// ---- GlobalTextList.TcGTLO
TEXTLIST GlobalTextList
  709 = ' abort_error.error_str_1: %s'
  714 = ' abort_error.error_str_2: %s'
  705 = ' abort_error.object_name: %s'
  8 = ' CASE PACKER SHIFT REGISTERS'
  724 = ' g_application_status: %s'
  719 = ' local_ams_net_id: %s'
  1320 = ' Number Of Tasks : %i'
  1337 = ' Online Change Count : %i'
  1311 = ' Project Name : %s  '
  1328 = ' Run Time n. : %i'
  424 = '%d'
  129 = '%dxd'
  192 = '%i Insert the error to simulate'
  334 = '%i Time Exceeded'
  1303 = '%iµS [MAX]'
  1345 = '%iµS [MIN]'
  83 = '%s'
  982 = '%s Insert the error to simulate'
  247 = '1st layer robot ID'
  249 = '2nd layer robot ID'
  252 = '3rd layer robot ID'
  254 = '4th layer robot ID'
  256 = '5th layer robot ID'
  710 = '6th layer robot ID'
  677 = '< Move'
  9 = 'ACC U CHANGE'
  1429 = 'ACCU COMPLETE'
  233 = 'ACCU START POSITION REQ'
  1537 = 'ACCU START REQ'
  470 = 'Actual error: %d mm'
  694 = 'Actual error: %s mm'
  344 = 'AFL codename  %s'
  337 = 'AFL date  %s'
  339 = 'AFL version  %s'
  81 = 'aHMI present'
  78 = 'aHMI version  %s'
  663 = 'Back Stop'
  929 = 'Belts'
  317 = 'CARTESIAN MODE'
  574 = 'Carton @\nBackstop'
  181 = 'CARTON ALIGNMENT'
  415 = 'CARTON DATA MATRIX'
  921 = 'CARTON FORMING SHIFT'
  42 = 'CARTON PICKUP SHIFT'
  496 = 'Case FC Lower LS PE Covered'
  498 = 'Case FC Lower OS PE Covered'
  497 = 'Case FC Upper LS PE Covered'
  499 = 'Case FC Upper OS PE Covered'
  707 = 'Case Fed'
  1245 = 'Case Loaded'
  919 = 'Case Open Flap LS PE Covered'
  928 = 'Case Open Flap OS PE Covered'
  713 = 'Case Present'
  902 = 'Case Reject PE Status'
  675 = 'Copy >'
  77 = 'CPU Load: %i %%'
  341 = 'CPU Temp: %i °C'
  577 = 'Crosspush\nREJECT'
  575 = 'Crosspush\nRequest'
  212 = 'CUPS FEEDING SHIFT'
  572 = 'Downstream\nRedefine'
  253 = 'Downstream Backup PE Covered'
  127 = 'drum equipment'
  579 = 'dsgdd'
  581 = 'E-Stop CLOSE'
  580 = 'E-Stop OPEN'
  321 = 'Elbow: %.3f deg'
  786 = 'Emergency'
  892 = 'Emergency CLOSE'
  560 = 'Emergency CLOSED'
  342 = 'Emergency OPEN'
  495 = 'Flap Detect Photoeyes'
  466 = 'forming equipment'
  1218 = 'Glue LS Upper Flap present'
  1263 = 'Glue OS Upper Flap present'
  423 = 'has 1st layer'
  237 = 'has 2nd layer'
  239 = 'has 3rd layer'
  241 = 'has 4th layer'
  243 = 'has 5th layer'
  245 = 'has 6th layer'
  881 = 'has carton'
  809 = 'has cup'
  149 = 'has glue'
  259 = 'INCOHERENT'
  79 = 'INITIAL CONFIGURATION\n(to set before PLC Run)'
  615 = 'INNER'
  987 = 'INNER\nMISALIGNMENT'
  735 = 'Insert the error to simulate'
  6 = 'Insert the error to simulate %i'
  730 = 'Insert the error to simulate: %s mm'
  578 = 'iPhysics'
  451 = 'item rejected'
  712 = 'item to be rejected'
  513 = 'JAM'
  320 = 'JOG MINUS'
  319 = 'JOG PLUS'
  316 = 'JOINT MODE'
  469 = 'LEFT LOWER'
  343 = 'LEFT UPPER'
  508 = 'Load'
  1294 = 'load %iµS -'
  803 = 'Lower left side sensor'
  158 = 'LOWER LEFT SIDE SENSOR'
  358 = 'LOWER RIGHT SIDE SENSOR'
  1190 = 'LS Lower Flap  present'
  1227 = 'LS Open Flap  present'
  1181 = 'LS Upper Flap  present'
  829 = 'MAX'
  370 = 'MESSAGE_ aHMI_Yellow OFF'
  665 = 'MESSAGE_ aHMI_Yellow_OFF'
  845 = 'MESSAGE_aHMI_Yellow_OFF'
  384 = 'MESSAGE_aHMI_Yellow_ON'
  173 = 'MIN'
  570 = 'Move Test'
  996 = 'NOMINAL'
  936 = 'Open Flap Eyes'
  576 = 'Open Guard'
  1208 = 'OS Lower Flap  present'
  1236 = 'OS Open Flap  present'
  1199 = 'OS Upper Flap  present'
  386 = 'OUTER\nMISALIGNMENT'
  676 = 'Phase Pos: %.3f deg'
  870 = 'Phase Pos: %.3f mm'
  318 = 'PHASE REQUEST'
  992 = 'PICK CARTONS'
  822 = 'PRODUCT\nABSENCE'
  183 = 'product ID'
  251 = 'Reject Backup PE Covered'
  248 = 'Reject Present PE Covered'
  569 = 'reject reason'
  945 = 'Reject Trigger PE Covered'
  151 = 'RESET'
  652 = 'RFID'
  394 = 'RIGHT LOWER'
  3 = 'RIGHT UPPER'
  255 = 'Robot Feed'
  974 = 'Robot ID'
  80 = 'selysionare la configurazione prima di mettere RUN il PLC'
  511 = 'Shoulder: %.3f deg'
  257 = 'SHUTTLE TOGGLE'
  910 = 'Simulate Load'
  755 = 'SIMULATION EMERGENCY BUTTON'
  953 = 'SIMULATION EMERGENCY BUTTON - CASE'
  887 = 'SIMULATION EMERGENCY BUTTON - TRANSFER'
  692 = 'SIMULATION EYBOARD'
  154 = 'SIMULATION KEYBOARD'
  322 = 'Speed: %.0f deg/s'
  515 = 'Speed: %.0f mm/s'
  153 = 'START'
  169 = 'START Sim - aHMI aperto'
  674 = 'step'
  509 = 'Step 1'
  516 = 'Step 2'
  518 = 'Step 3'
  893 = 'Step 4'
  152 = 'STOP'
  700 = 'Task monitor'
  872 = 'Tilt: %.3f deg'
  1254 = 'Transfer SR1'
  61 = 'UNDER_MIN'
  464 = 'UPPER LEFT SIDE SENSOR'
  202 = 'UPPER RIGHT SIDE SENSOR'
  573 = 'Upstack\nTest\nMode'
  571 = 'Upstream\nRedefine'
  82 = 'Video presente e collegato'
  512 = 'Wrist: %.3f deg'
  514 = 'X: %.3f mm'
  871 = 'Y: %.3f mm'
  88 = 'Yellow Message OFF'
  771 = 'Yellow Message ON'
  729 = '[1] highest %iµS - '
  734 = '[2] norm %iµS - '
  1277 = '[3] low %iµS - '
  1286 = '[4] lowest %iµS - '
END_TEXTLIST

// ---- Visualization/AFL/VISU_MAIN.TcVIS
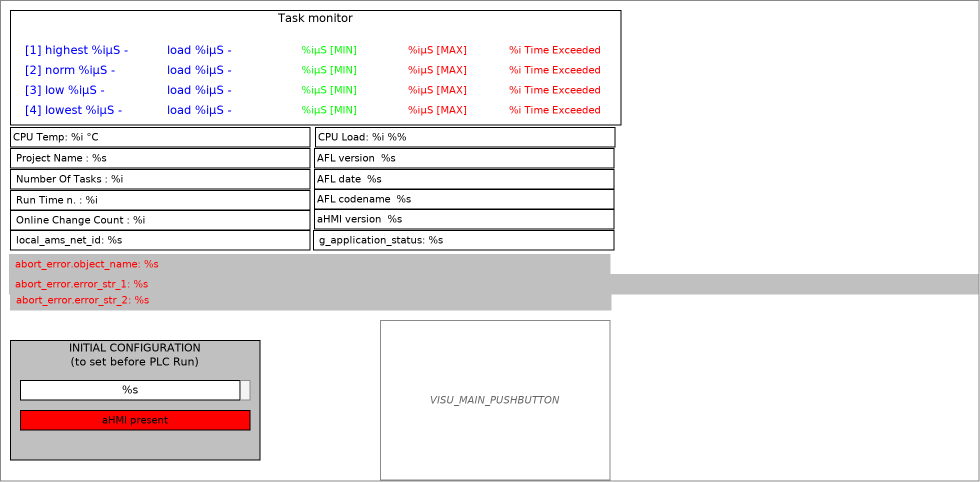
VISUALIZATION VISU_MAIN  // 980x482
    Rectangle (10,10 611x115), "Task monitor"
    Rectangle (9,254 601x20), "abort_error.object_name: %s", text variable: abort_error.object_name
    Rectangle (9,274 969x20), "abort_error.error_str_1: %s", text variable: abort_error.error_str_1
    Rectangle (10,290 601x20), "abort_error.error_str_2: %s", text variable: abort_error.error_str_2
    Rectangle (10,230 300x20), "local_ams_net_id: %s", text variable: local_ams_net_id
    Rectangle (313,230 301x20), "g_application_status: %s", text variable: Application_Common.g_application_status
    Rectangle (22,40 130x20), "[1] highest %iµS -", text variable: afl_tasks[1].cycle_us
    Rectangle (22,60 130x20), "[2] norm %iµS -", text variable: afl_tasks[2].cycle_us
    Rectangle (22,80 130x20), "[3] low %iµS -", text variable: afl_tasks[3].cycle_us
    Rectangle (22,100 130x20), "[4] lowest %iµS -", text variable: afl_tasks[4].cycle_us
    Rectangle (164,100 100x20), "load %iµS -", text variable: afl_tasks[4].task_profiler_data.AverageExecTime
    Rectangle (164,80 100x20), "load %iµS -", text variable: afl_tasks[3].task_profiler_data.AverageExecTime
    Rectangle (164,60 100x20), "load %iµS -", text variable: afl_tasks[2].task_profiler_data.AverageExecTime
    Rectangle (164,40 100x20), "load %iµS -", text variable: afl_tasks[1].task_profiler_data.AverageExecTime
    Rectangle (380,40 90x20), "%iµS [MAX]", text variable: afl_tasks[1].task_profiler_data.MaxExecTime
    Rectangle (380,60 90x20), "%iµS [MAX]", text variable: afl_tasks[2].task_profiler_data.MaxExecTime
    Rectangle (380,80 90x20), "%iµS [MAX]", text variable: afl_tasks[2].task_profiler_data.MaxExecTime
    Rectangle (380,100 90x20), "%iµS [MAX]", text variable: afl_tasks[4].task_profiler_data.MaxExecTime
    Rectangle (10,148 300x20), "Project Name : %s", text variable: SystemInfo.projectName
    Rectangle (10,169 300x20), "Number Of Tasks : %i", text variable: SystemInfo.numberOfTasks
    Rectangle (10,190 300x20), "Run Time n. : %i", text variable: SystemInfo.runTimeNo
    Rectangle (10,210 300x20), "Online Change Count : %i", text variable: SystemInfo.onlineChangeCount
    Rectangle (250,100 110x20), "%iµS [MIN]", text variable: afl_tasks[4].task_profiler_data.MinExecTime
    Rectangle (250,80 110x20), "%iµS [MIN]", text variable: afl_tasks[3].task_profiler_data.MinExecTime
    Rectangle (250,60 110x20), "%iµS [MIN]", text variable: afl_tasks[2].task_profiler_data.MinExecTime
    Rectangle (250,40 110x20), "%iµS [MIN]", text variable: afl_tasks[1].task_profiler_data.MinExecTime
    Rectangle (506,40 110x20), "%i Time Exceeded", text variable: SystemTaskInfoArr[1].cycleTimeExceeded
    Rectangle (506,60 110x20), "%i Time Exceeded", text variable: SystemTaskInfoArr[2].cycleTimeExceeded
    Rectangle (506,80 110x20), "%i Time Exceeded", text variable: SystemTaskInfoArr[3].cycleTimeExceeded
    Rectangle (506,100 110x20), "%i Time Exceeded", text variable: SystemTaskInfoArr[4].cycleTimeExceeded
    Rectangle (314,169 300x20), "AFL date %s", text variable: AFL_VERSION.v_date
    Rectangle (314,148 300x20), "AFL version %s", text variable: AFL_VERSION.s_value
    Rectangle (10,127 300x20), "CPU Temp: %i °C", text variable: .system_diagnosis.cpu_temperature_actual_value
    Rectangle (314,189 300x20), "AFL codename %s", text variable: AFL_VERSION.development_stage
    Rectangle (315,127 300x20), "CPU Load: %i %%", text variable: system_diagnosis.cpu_usage_actual_value
    Rectangle (314,209 300x20), "aHMI version %s", text variable: hmi.private.major_version
    Frame (380,320 230x160)
        shows VISU_MAIN_PUSHBUTTON(m_Input_mch := EZ.mch, m_Input_stop := ez_mch_services_pushbuttons_main.stop_button_di, m_Input_reset := ez_mch_services_pushbuttons_main.reset_button_di, m_Input_start := ez_mch_services_pushbuttons_main.start_button_pressed_di)
    Rectangle (10,340 250x120), "INITIAL CONFIGURATION (to set before PLC Run)", tooltip "selysionare la configurazione prima di mettere RUN il PLC"
    RoundedRectangle (20,410 230x20), "aHMI present", tooltip "Video presente e collegato", colour toggle: Application_Common.HMI_IS_REQUIRED_DVR
        toggle Application_Common.HMI_IS_REQUIRED_DVR
    RoundedRectangle (20,380 220x20), "%s", text variable: .test_target_device
    Scrollbar (240,380 10x20)
        p1057716461: .test_target_device
END_VISUALIZATION

// ---- Visualization/Carton feeding/CARTON_FEEDING_TOOTH_DISTANCE.TcVIS
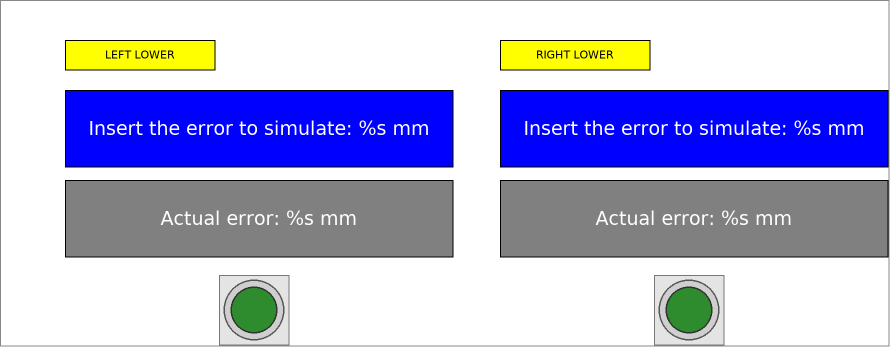
VISUALIZATION CARTON_FEEDING_TOOTH_DISTANCE  // 890x347
    Rectangle (65,40 150x30), "LEFT LOWER"
    Rectangle (500,40 150x30), "RIGHT LOWER"
    RoundedRectangle (65,90 388x77), "Insert the error to simulate: %s mm", text variable: wu_cartonFeeding_leftSide_toothDistance.simulation_error
        OnMouseUp: write the text variable via VisuDialogs.Numpad
    RoundedRectangle (500,90 388x77), "Insert the error to simulate: %s mm", text variable: wu_cartonFeeding_rightSide_toothDistance.simulation_error
        OnMouseUp: write the text variable via VisuDialogs.Numpad
    RoundedRectangle (65,180 388x77), "Actual error: %s mm", text variable: wu_cartonFeeding_leftSide_toothDistance.simulation_error_current_value_visu
        OnMouseUp: write the text variable via VisuDialogs.Numpad
    RoundedRectangle (500,180 388x77), "Actual error: %s mm", text variable: wu_cartonFeeding_rightSide_toothDistance.simulation_error_current_value_visu
        OnMouseUp: write the text variable via VisuDialogs.Numpad
    PushSwitch (219,275 70x70), variable: wu_cartonFeeding_leftSide_toothDistance.simulation_error_download, behaviour: TAP, style: Switch-PushSwitch-Green
    PushSwitch (654,275 70x70), variable: wu_cartonFeeding_rightSide_toothDistance.simulation_error_download, behaviour: TAP, style: Switch-PushSwitch-Green
END_VISUALIZATION

// ---- Visualization/Carton forming/CARTON_FORMING_CHECKS.TcVIS
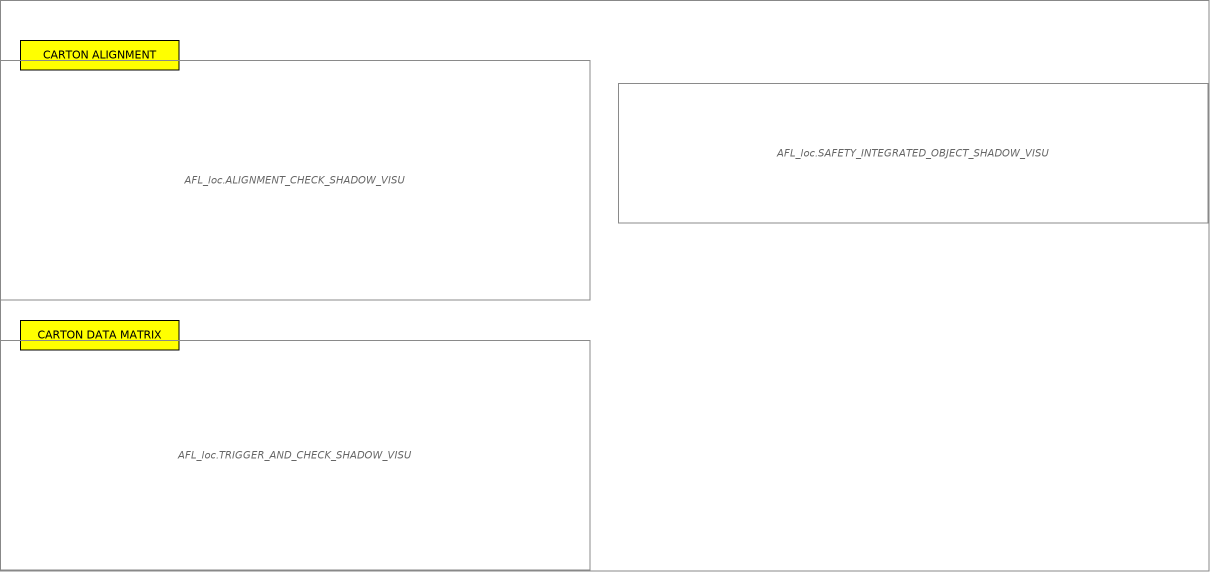
VISUALIZATION CARTON_FORMING_CHECKS  // 1210x572
    Rectangle (20,40 159x30), "CARTON ALIGNMENT"
    Frame (0,60 590x240)
        shows AFL_loc.ALIGNMENT_CHECK_SHADOW_VISU(m_Input_alignment_check_shadow := dbg_wu_cartonforming_belt_checks.algnchk_shd)
    Rectangle (20,320 159x30), "CARTON DATA MATRIX"
    Frame (0,340 590x230)
        shows AFL_loc.TRIGGER_AND_CHECK_SHADOW_VISU(m_Input_trigger_and_check_shadow := dbg_wu_cartonforming_belt_checks.data_matrix_tchk_shd)
    Frame (618,83 590x140)
        shows AFL_loc.SAFETY_INTEGRATED_OBJECT_SHADOW_VISU(m_Input_safety_integrated_object_shadow := dbg_wu_main_safety_guards.sio_shd)
END_VISUALIZATION

// ---- Visualization/Casepacker_Keyboard.TcVIS
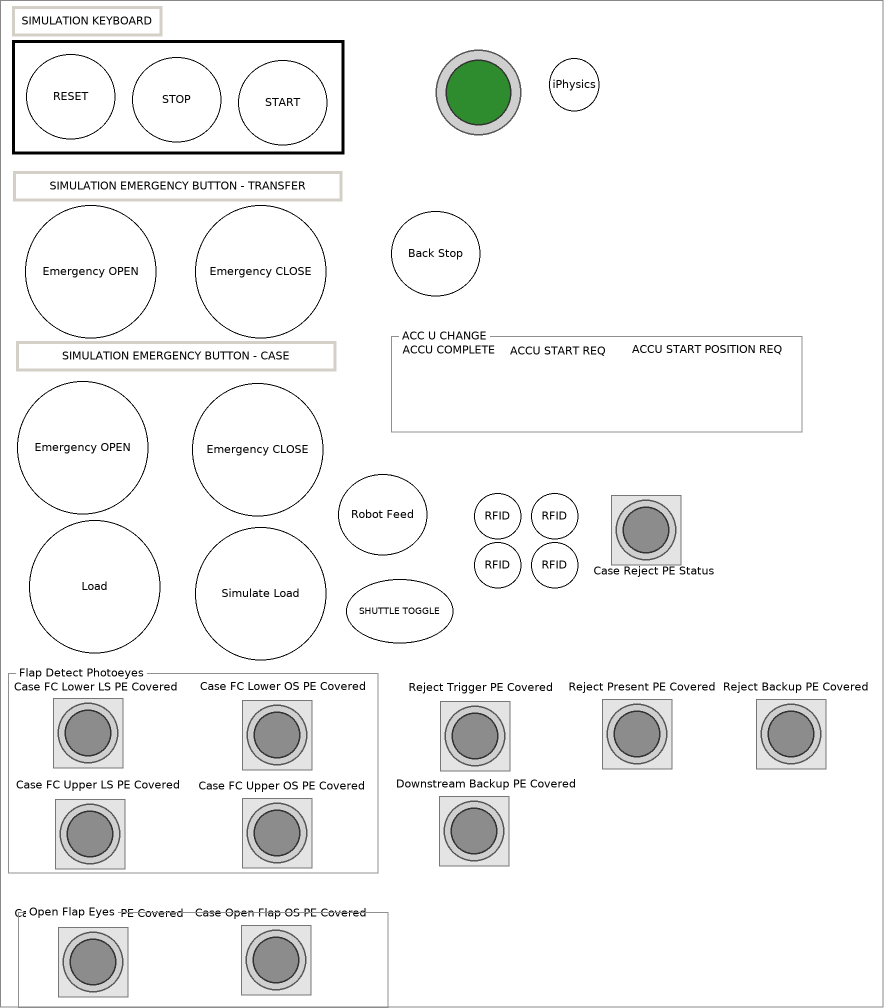
VISUALIZATION Casepacker_Keyboard  // 884x1008
    Rectangle (12,40 332x114)
    Ellipse (26,54 89x85), "RESET"
        tap csp_transfer_main_services_pushbuttons.visu_reset
    Ellipse (132,57 89x85), "STOP"
        tap csp_transfer_main_services_pushbuttons.visu_stop
    Ellipse (238,60 89x85), "START"
        tap csp_transfer_main_services_pushbuttons.visu_start
    Textfield (12,6 150x30), "SIMULATION KEYBOARD"
    Ellipse (25,205 131x133), "Emergency OPEN"
        tap csp_transfer_main_services_pushbuttons.visu_emergency_open
    Ellipse (195,205 131x133), "Emergency CLOSE"
        tap csp_transfer_main_services_pushbuttons.visu_emergency_close
    Textfield (13,171 329x30), "SIMULATION EMERGENCY BUTTON - TRANSFER"
    Lamp1 (426,43 105x99), variable: csp_transfer_main_safety_emergency.HMI_button_lamp_do.field.status, style: Lamp-Lamp1-Green
    Ellipse (391,211 89x85), "Back Stop", colour toggle: csp_transfer_upstacker_sensors.debug_carton_backstop
        toggle csp_transfer_upstacker_sensors.debug_carton_backstop
    Ellipse (192,383 131x133), "Emergency CLOSE"
        tap csp_case_main_services_pushbuttons.visu_emergency_close
    Textfield (16,341 320x30), "SIMULATION EMERGENCY BUTTON - CASE"
    Ellipse (17,381 131x133), "Emergency OPEN"
        tap csp_case_main_services_pushbuttons.visu_emergency_open
    Ellipse (549,58 50x53), "iPhysics"
        toggle MAIN.IP_enable
    GroupBox (8,665 370x208), "Flap Detect Photoeyes"
        PushSwitchLed (45,33 70x70), variable: dbg_csp_case_fc_ls_lower_sensors.flap_chksect_shd.force_input_status, behaviour: TOGGLE, style: Switch-PushSwitchLed-Gray
    Ellipse (29,520 131x133), "Load"
        tap csp_case_loader.load_request
    Ellipse (531,493 47x46), "RFID"
        toggle csp_case_closing_ls_upper.rfid_fake
    Ellipse (531,542 47x46), "RFID"
        toggle csp_case_closing_ls_lower.rfid_fake
    Ellipse (474,493 47x46), "RFID"
        toggle csp_case_closing_os_upper.rfid_fake
    Ellipse (474,542 47x46), "RFID"
        toggle csp_case_closing_os_lower.rfid_fake
    PushSwitchLed (611,495 70x70), behaviour: TOGGLE, style: Switch-PushSwitchLed-Gray
    Label (579,556 150x30), "Case Reject PE Status"
    Ellipse (195,527 131x133), "Simulate Load"
        tap csp_case_transport.product_loaded
    Label (8,673 176x28), "Case FC Lower LS PE Covered"
    PushSwitchLed (55,799 70x70), variable: dbg_csp_case_fc_ls_upper_sensors.flap_chksect_shd.force_input_status, behaviour: TOGGLE, style: Switch-PushSwitchLed-Gray
    Label (10,775 176x20), "Case FC Upper LS PE Covered"
    PushSwitchLed (242,700 70x70), variable: dbg_csp_case_fc_os_lower_sensors.flap_chksect_shd.force_input_status, behaviour: TOGGLE, style: Switch-PushSwitchLed-Gray
    Label (195,678 176x17), "Case FC Lower OS PE Covered"
    PushSwitchLed (242,798 70x70), variable: dbg_csp_case_fc_os_upper_sensors.flap_chksect_shd.force_input_status, behaviour: TOGGLE, style: Switch-PushSwitchLed-Gray
    Label (194,777 176x18), "Case FC Upper OS PE Covered"
    Label (8,888 176x28)
    PushSwitchLed (58,927 70x70), variable: dbg_csp_case_openflap_sensors.open_flap_ls_di_dchk_shd.force_input_status, behaviour: TOGGLE, style: Switch-PushSwitchLed-Gray
    Label (11,905 176x17), "Case Open Flap LS PE Covered"
    PushSwitchLed (241,925 70x70), variable: dbg_csp_case_openflap_sensors.open_flap_os_di_dchk_shd.force_input_status, behaviour: TOGGLE, style: Switch-PushSwitchLed-Gray
    Label (193,904 176x18), "Case Open Flap OS PE Covered"
    GroupBox (391,328 411x104), "ACC U CHANGE"
        Label (381,-232 176x28)
        Label (79,9 176x28), "ACCU START REQ"
    PushSwitchLed (440,701 70x70), variable: dbg_csp_case_discharge_reject_sensors.reject_trigger_inchoerence_chksect_shd.force_input_status, behaviour: TOGGLE, style: Switch-PushSwitchLed-Gray
    Label (393,679 176x17), "Reject Trigger PE Covered"
    PushSwitchLed (602,699 70x70), variable: dbg_csp_case_discharge_reject_sensors.reject_present_di_shd.is_covered, behaviour: TOGGLE, style: Switch-PushSwitchLed-Gray
    Label (554,678 176x18), "Reject Present PE Covered"
    PushSwitchLed (756,699 70x70), variable: dbg_csp_case_discharge_reject_sensors.reject_backup_di_shd.is_covered, behaviour: TOGGLE, style: Switch-PushSwitchLed-Gray
    Label (708,678 176x18), "Reject Backup PE Covered"
    PushSwitchLed (439,796 70x70), variable: dbg_csp_case_discharge_reject_sensors.downstream_backup_di_shd.is_covered, behaviour: TOGGLE, style: Switch-PushSwitchLed-Gray
    Label (391,775 190x18), "Downstream Backup PE Covered"
    Ellipse (338,474 89x81), "Robot Feed"
        toggle csp_case_feed.Feed_request
    Ellipse (346,579 107x64), "SHUTTLE TOGGLE"
        toggle csp_case_transport.product_loaded
    GroupBox (18,904 370x104), "Open Flap Eyes"
        Label (381,-232 176x28)
    Label (361,336 176x28), "ACCU COMPLETE"
    Label (619,327 176x45), "ACCU START POSITION REQ"
END_VISUALIZATION

// ---- Visualization/cp_visu/Visualization_1.TcVIS
VISUALIZATION Visualization_1  // 2x2
END_VISUALIZATION

// ---- Visualization/CSP_Case_Feed_Kinematic.TcVIS
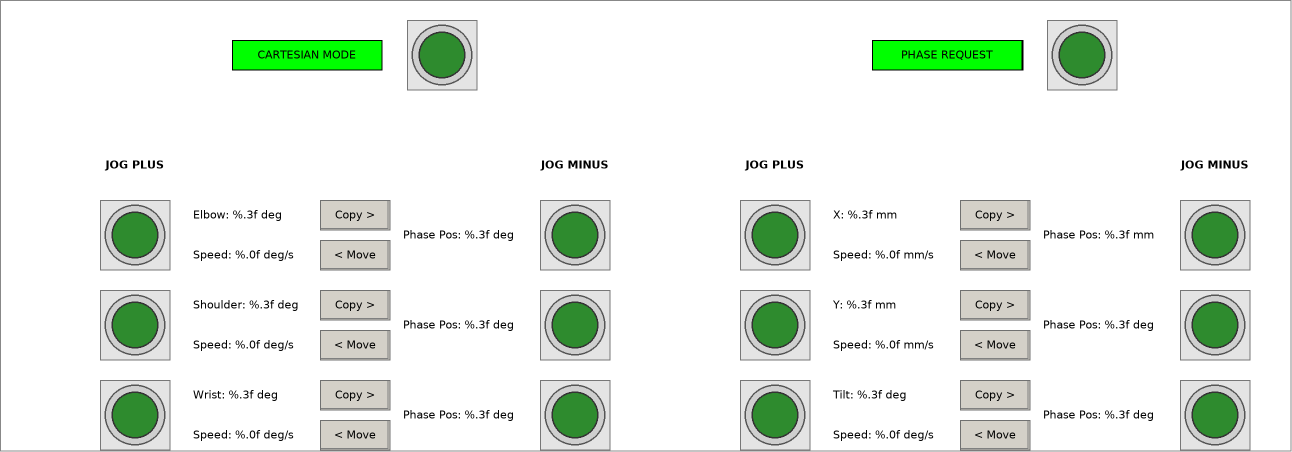
VISUALIZATION CSP_Case_Feed_Kinematic  // 1292x452
    Group (232,20 245x70)
        Rectangle (0,20 150x30), "JOINT MODE", invisible if: csp_case_feed_kinematic.kin_config_cartesian_mode
        PushSwitch (175,0 70x70), variable: csp_case_feed_kinematic.joint_cartesian_mode, input disabled if: csp_case_feed_kinematic.visu_disable_general_command, behaviour: TAP, style: Switch-PushSwitch-Green
        Rectangle (0,20 150x30), "CARTESIAN MODE", invisible if: not csp_case_feed_kinematic.kin_config_cartesian_mode
    Group (872,20 245x70)
        Rectangle (1,20 150x30), "PHASE REQUEST", invisible if: csp_case_feed_kinematic.phase_request
        PushSwitch (175,0 70x70), variable: csp_case_feed_kinematic.phase_request, input disabled if: csp_case_feed_kinematic.visu_disable_phase_request, behaviour: TOGGLE, style: Switch-PushSwitch-Green
        Rectangle (0,20 150x30), "PHASE REQUEST", invisible if: not csp_case_feed_kinematic.phase_request
    Rectangle (60,150 150x30), "JOG PLUS"
    Rectangle (500,150 150x30), "JOG MINUS"
    Group (100,200 510x70)
        Rectangle (90,0 140x30), "Elbow: %.3f deg", text variable: csp_case_feed_kinematic.elbow_actual_position
        PushSwitch (0,0 70x70), variable: csp_case_feed_kinematic.elbow_jog_plus, input disabled if: csp_case_feed_kinematic.visu_disable_ACS_jog_mode, behaviour: TAP, style: Switch-PushSwitch-Green
        PushSwitch (440,0 70x70), variable: csp_case_feed_kinematic.elbow_jog_minus, input disabled if: csp_case_feed_kinematic.visu_disable_ACS_jog_mode, behaviour: TAP, style: Switch-PushSwitch-Green
        Rectangle (90,40 140x30), "Speed: %.0f deg/s", text variable: csp_case_feed_kinematic.elbow_move_speed
            OnMouseDown: write csp_case_feed_kinematic.elbow_move_speed via VisuDialogs.Numpad, min 0, max 100, format %.0f
        Button (220,0 70x30), "Copy >", input disabled if: csp_case_feed_kinematic.visu_disable_ACS_command
            tap csp_case_feed_kinematic.elbow_copy_phase
        Rectangle (300,20 140x30), "Phase Pos: %.3f deg", text variable: csp_case_feed_kinematic.elbow_phase_position
            OnMouseDown: write csp_case_feed_kinematic.elbow_phase_position via VisuDialogs.Numpad, min -200, max 200, format %.3f
        Button (220,40 70x30), "< Move", input disabled if: csp_case_feed_kinematic.visu_disable_ACS_command
            tap csp_case_feed_kinematic.elbow_phase_move
    Group (100,290 510x70)
        Rectangle (90,0 140x30), "Shoulder: %.3f deg", text variable: csp_case_feed_kinematic.shoulder_actual_position
        PushSwitch (0,0 70x70), variable: csp_case_feed_kinematic.shoulder_jog_plus, input disabled if: csp_case_feed_kinematic.visu_disable_ACS_jog_mode, behaviour: TAP, style: Switch-PushSwitch-Green
        PushSwitch (440,0 70x70), variable: csp_case_feed_kinematic.shoulder_jog_minus, input disabled if: csp_case_feed_kinematic.visu_disable_ACS_jog_mode, behaviour: TAP, style: Switch-PushSwitch-Green
        Rectangle (90,40 140x30), "Speed: %.0f deg/s", text variable: csp_case_feed_kinematic.shoulder_move_speed
            OnMouseDown: write csp_case_feed_kinematic.shoulder_move_speed via VisuDialogs.Numpad, min 0, max 100, format %.0f
        Button (220,0 70x30), "Copy >", input disabled if: csp_case_feed_kinematic.visu_disable_ACS_command
            tap csp_case_feed_kinematic.shoulder_copy_phase
        Rectangle (300,20 140x30), "Phase Pos: %.3f deg", text variable: csp_case_feed_kinematic.shoulder_phase_position
            OnMouseDown: write csp_case_feed_kinematic.shoulder_phase_position via VisuDialogs.Numpad, min -200, max 200, format %.3f
        Button (220,40 70x30), "< Move", input disabled if: csp_case_feed_kinematic.visu_disable_ACS_command
            tap csp_case_feed_kinematic.shoulder_phase_move
    Group (100,380 510x70)
        Rectangle (90,0 140x30), "Wrist: %.3f deg", text variable: csp_case_feed_kinematic.wrist_actual_position
        PushSwitch (0,0 70x70), variable: csp_case_feed_kinematic.wrist_jog_plus, input disabled if: csp_case_feed_kinematic.visu_disable_ACS_jog_mode, behaviour: TAP, style: Switch-PushSwitch-Green
        PushSwitch (440,0 70x70), variable: csp_case_feed_kinematic.wrist_jog_minus, input disabled if: csp_case_feed_kinematic.visu_disable_ACS_jog_mode, behaviour: TAP, style: Switch-PushSwitch-Green
        Rectangle (90,40 140x30), "Speed: %.0f deg/s", text variable: csp_case_feed_kinematic.wrist_move_speed
            OnMouseDown: write csp_case_feed_kinematic.wrist_move_speed via VisuDialogs.Numpad, min 0, max 100, format %.0f
        Button (220,0 70x30), "Copy >", input disabled if: csp_case_feed_kinematic.visu_disable_ACS_command
            tap csp_case_feed_kinematic.wrist_copy_phase
        Rectangle (300,20 140x30), "Phase Pos: %.3f deg", text variable: csp_case_feed_kinematic.wrist_phase_position
            OnMouseDown: write csp_case_feed_kinematic.wrist_phase_position via VisuDialogs.Numpad, min -200, max 200, format %.3f
        Button (220,40 70x30), "< Move", input disabled if: csp_case_feed_kinematic.visu_disable_ACS_command
            tap csp_case_feed_kinematic.wrist_phase_move
    Group (740,200 510x70)
        Rectangle (90,0 140x30), "X: %.3f mm", text variable: csp_case_feed_kinematic.x_actual_position
        PushSwitch (0,0 70x70), variable: csp_case_feed_kinematic.x_jog_plus, input disabled if: csp_case_feed_kinematic.visu_disable_MCS_jog_mode, behaviour: TAP, style: Switch-PushSwitch-Green
        PushSwitch (440,0 70x70), variable: csp_case_feed_kinematic.x_jog_minus, input disabled if: csp_case_feed_kinematic.visu_disable_MCS_jog_mode, behaviour: TAP, style: Switch-PushSwitch-Green
        Rectangle (90,40 140x30), "Speed: %.0f mm/s", text variable: csp_case_feed_kinematic.x_move_speed
            OnMouseDown: write csp_case_feed_kinematic.x_move_speed via VisuDialogs.Numpad, min 0, max 100, format %.0f
        Button (220,0 70x30), "Copy >", input disabled if: csp_case_feed_kinematic.visu_disable_MCS_command
            tap csp_case_feed_kinematic.x_copy_phase
        Rectangle (300,20 140x30), "Phase Pos: %.3f mm", text variable: csp_case_feed_kinematic.x_phase_position
            OnMouseDown: write csp_case_feed_kinematic.x_phase_position via VisuDialogs.Numpad, min -2000, max 2000, format %.3f
        Button (220,40 70x30), "< Move", input disabled if: csp_case_feed_kinematic.visu_disable_MCS_command
            tap csp_case_feed_kinematic.x_phase_move
    Rectangle (1140,150 150x30), "JOG MINUS"
    Rectangle (700,150 150x30), "JOG PLUS"
    Group (740,290 510x70)
        Rectangle (90,0 140x30), "Y: %.3f mm", text variable: csp_case_feed_kinematic.y_actual_position
        PushSwitch (0,0 70x70), variable: csp_case_feed_kinematic.y_jog_plus, input disabled if: csp_case_feed_kinematic.visu_disable_MCS_jog_mode, behaviour: TAP, style: Switch-PushSwitch-Green
        PushSwitch (440,0 70x70), variable: csp_case_feed_kinematic.y_jog_minus, input disabled if: csp_case_feed_kinematic.visu_disable_MCS_jog_mode, behaviour: TAP, style: Switch-PushSwitch-Green
        Rectangle (90,40 140x30), "Speed: %.0f mm/s", text variable: csp_case_feed_kinematic.y_move_speed
            OnMouseDown: write csp_case_feed_kinematic.y_move_speed via VisuDialogs.Numpad, min 0, max 100, format %.0f
        Button (220,0 70x30), "Copy >", input disabled if: csp_case_feed_kinematic.visu_disable_MCS_command
            tap csp_case_feed_kinematic.y_copy_phase
        Rectangle (300,20 140x30), "Phase Pos: %.3f deg", text variable: csp_case_feed_kinematic.y_phase_position
            OnMouseDown: write csp_case_feed_kinematic.y_phase_position via VisuDialogs.Numpad, min -100, max 1000, format %.3f
        Button (220,40 70x30), "< Move", input disabled if: csp_case_feed_kinematic.visu_disable_MCS_command
            tap csp_case_feed_kinematic.y_phase_move
    Group (740,380 510x70)
        Rectangle (90,0 140x30), "Tilt: %.3f deg", text variable: csp_case_feed_kinematic.tilt_actual_position
        PushSwitch (0,0 70x70), variable: csp_case_feed_kinematic.tilt_jog_plus, input disabled if: csp_case_feed_kinematic.visu_disable_MCS_jog_mode, behaviour: TAP, style: Switch-PushSwitch-Green
        PushSwitch (440,0 70x70), variable: csp_case_feed_kinematic.tilt_jog_minus, input disabled if: csp_case_feed_kinematic.visu_disable_MCS_jog_mode, behaviour: TAP, style: Switch-PushSwitch-Green
        Rectangle (90,40 140x30), "Speed: %.0f deg/s", text variable: csp_case_feed_kinematic.tilt_move_speed
            OnMouseDown: write csp_case_feed_kinematic.tilt_move_speed via VisuDialogs.Numpad, min 0, max 100, format %.0f
        Button (220,0 70x30), "Copy >", input disabled if: csp_case_feed_kinematic.visu_disable_MCS_command
            tap csp_case_feed_kinematic.tilt_copy_phase
        Rectangle (300,20 140x30), "Phase Pos: %.3f deg", text variable: csp_case_feed_kinematic.tilt_phase_position
            OnMouseDown: write csp_case_feed_kinematic.tilt_phase_position via VisuDialogs.Numpad, min 0, max 150, format %.3f
        Button (220,40 70x30), "< Move", input disabled if: csp_case_feed_kinematic.visu_disable_MCS_command
            tap csp_case_feed_kinematic.tilt_phase_move
END_VISUALIZATION

// ---- Visualization/Transfer_Keyboard.TcVIS
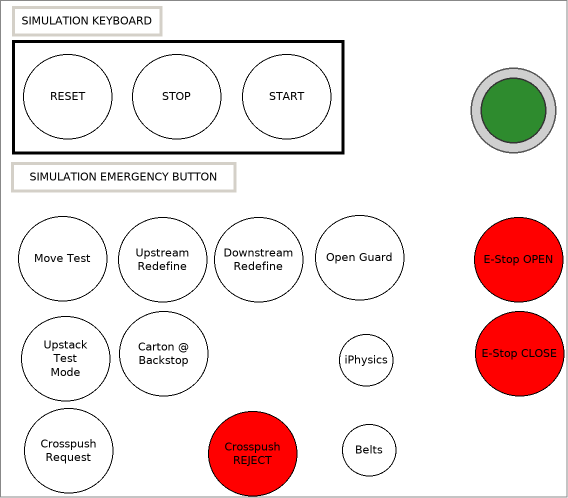
VISUALIZATION Transfer_Keyboard  // 568x498
    Rectangle (12,40 332x114)
    Ellipse (23,54 89x85), "RESET"
        tap csp_transfer_main_services_pushbuttons.visu_reset
    Ellipse (132,54 89x85), "STOP"
        tap csp_transfer_main_services_pushbuttons.visu_stop
    Ellipse (242,54 89x85), "START"
        tap csp_transfer_main_services_pushbuttons.visu_start
    Textfield (12,6 150x30), "SIMULATION KEYBOARD"
    Textfield (11,162 225x30), "SIMULATION EMERGENCY BUTTON"
    Lamp1 (461,61 105x99), variable: csp_transfer_main_safety_emergency.HMI_button_lamp_do.field.status, style: Lamp-Lamp1-Green
    Ellipse (18,216 89x85), "Move Test"
        toggle csp_transfer_upstacker_virtualMaster.move_test_enable
    Ellipse (118,217 89x85), "Upstream Redefine"
        tap csp_transfer_upstacker_virtualMaster.move_test_redefine_upstream
    Ellipse (214,217 89x85), "Downstream Redefine"
        tap csp_transfer_upstacker_virtualMaster.move_test_redefine_downstream
    Ellipse (21,316 89x85), "Upstack Test Mode"
        toggle csp_transfer_upstacker_sensors.debug_active
    Ellipse (119,311 89x85), "Carton @ Backstop"
        toggle csp_transfer_upstacker_sensors.debug_carton_backstop
    Ellipse (24,408 89x85), "Crosspush Request"
        toggle csp_transfer_crosspusher.move_request
    Ellipse (315,215 89x85), "Open Guard"
        toggle csp_transfer_upstacker_virtualMaster.guard_open
    Ellipse (208,411 89x85), "Crosspush REJECT"
        tap csp_transfer_crosspusher_sensors.reject_stack
    Ellipse (339,334 54x52), "iPhysics"
        toggle IP_Main.IP_enable
    Ellipse (474,217 89x85), "E-Stop OPEN"
        tap csp_case_main_services_pushbuttons.visu_emergency_open
    Ellipse (475,311 89x85), "E-Stop CLOSE"
        tap csp_case_main_services_pushbuttons.visu_emergency_close
    Ellipse (342,424 54x52), "Belts"
        toggle csp_transfer_infeed_clamp.start_infeed_belts
END_VISUALIZATION

// ---- Visualization/Shift register/Carton filling/CARTON_FILLING_SHIFT_ELEMENT.TcVIS
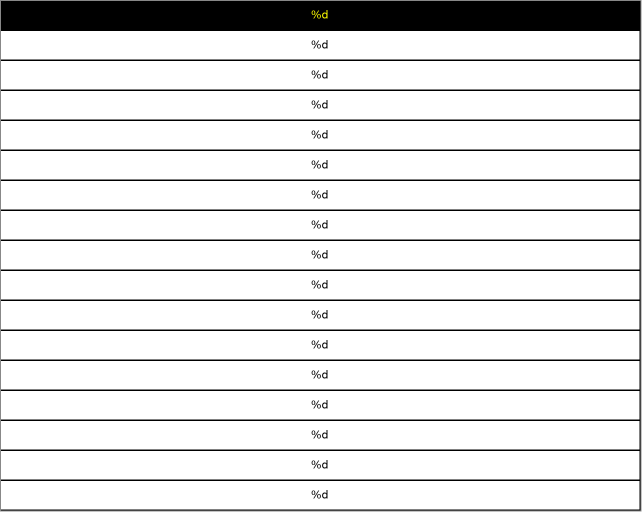
VISUALIZATION CARTON_FILLING_SHIFT_ELEMENT  // 642x512
VAR_INPUT
	index:		UDINT;
END_VAR
    Rectangle (0,0 640x30), "%d", text variable: wu_cartonForming_shiftRegister_debug.shift_debug[index].step_id
    Rectangle (0,30 640x30), "%d", text variable: wu_cartonFilling_shiftRegister_debug.shift_debug[index].status.0, colour toggle: wu_cartonFilling_shiftRegister_debug.shift_debug[index].status.0
    Rectangle (0,90 640x30), "%d", text variable: wu_cartonFilling_shiftRegister_debug.shift_debug[index].reject_reason
    Rectangle (0,120 640x30), "%d", text variable: wu_cartonFilling_shiftRegister_debug.shift_debug[index].status.4, colour toggle: wu_cartonFilling_shiftRegister_debug.shift_debug[index].status.4
    Rectangle (0,180 640x30), "%d", text variable: wu_cartonFilling_shiftRegister_debug.shift_debug[index].status.11, colour toggle: wu_cartonFilling_shiftRegister_debug.shift_debug[index].status.11
    Rectangle (0,150 640x30), "%d", text variable: wu_cartonFilling_shiftRegister_debug.shift_debug[index].status.10, colour toggle: wu_cartonFilling_shiftRegister_debug.shift_debug[index].status.10
    Rectangle (0,60 640x30), "%d", text variable: wu_cartonFilling_shiftRegister_debug.shift_debug[index].status.1, colour toggle: wu_cartonFilling_shiftRegister_debug.shift_debug[index].status.1
    Rectangle (0,210 640x30), "%d", text variable: wu_cartonFilling_shiftRegister_debug.shift_debug[index].status.12, colour toggle: wu_cartonFilling_shiftRegister_debug.shift_debug[index].status.12
    Rectangle (0,240 640x30), "%d", text variable: wu_cartonFilling_shiftRegister_debug.shift_debug[index].status.13, colour toggle: wu_cartonFilling_shiftRegister_debug.shift_debug[index].status.13
    Rectangle (0,270 640x30), "%d", text variable: wu_cartonFilling_shiftRegister_debug.shift_debug[index].status.14, colour toggle: wu_cartonFilling_shiftRegister_debug.shift_debug[index].status.14
    Rectangle (0,300 640x30), "%d", text variable: wu_cartonFilling_shiftRegister_debug.shift_debug[index].status.15, colour toggle: wu_cartonFilling_shiftRegister_debug.shift_debug[index].status.15
    Rectangle (0,330 640x30), "%d", text variable: wu_cartonFilling_shiftRegister_debug.shift_debug[index]._1st_layer_robot_id
    Rectangle (0,360 640x30), "%d", text variable: wu_cartonFilling_shiftRegister_debug.shift_debug[index]._2nd_layer_robot_id
    Rectangle (0,390 640x30), "%d", text variable: wu_cartonFilling_shiftRegister_debug.shift_debug[index]._3rd_layer_robot_id
    Rectangle (0,420 640x30), "%d", text variable: wu_cartonFilling_shiftRegister_debug.shift_debug[index]._4th_layer_robot_id
    Rectangle (0,450 640x30), "%d", text variable: wu_cartonFilling_shiftRegister_debug.shift_debug[index]._5th_layer_robot_id
    Rectangle (0,480 640x30), "%d", text variable: wu_cartonFilling_shiftRegister_debug.shift_debug[index]._6th_layer_robot_id
END_VISUALIZATION

// ---- Visualization/Shift register/Carton filling/CARTON_FILLING_SHIFT_ELEMENT_DESCRIPTION.TcVIS
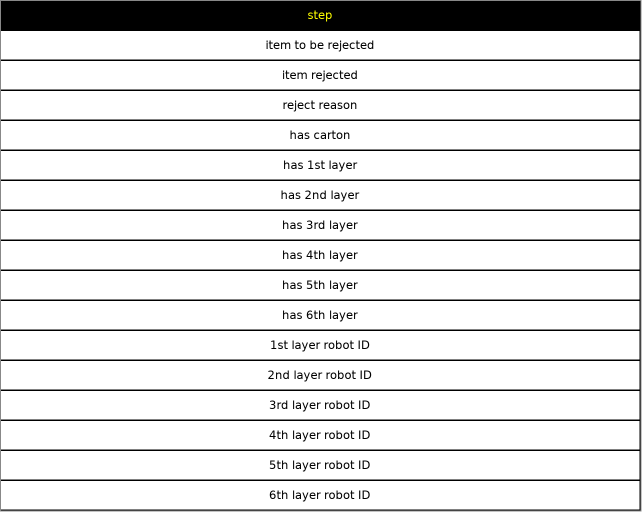
VISUALIZATION CARTON_FILLING_SHIFT_ELEMENT_DESCRIPTION  // 642x512
    Rectangle (0,0 640x30), "step"
    Rectangle (0,30 640x30), "item to be rejected"
    Rectangle (0,90 640x30), "reject reason"
    Rectangle (0,120 640x30), "has carton"
    Rectangle (0,150 640x30), "has 1st layer"
    Rectangle (0,60 640x30), "item rejected"
    Rectangle (0,180 640x30), "has 2nd layer"
    Rectangle (0,210 640x30), "has 3rd layer"
    Rectangle (0,240 640x30), "has 4th layer"
    Rectangle (0,270 640x30), "has 5th layer"
    Rectangle (0,300 640x30), "has 6th layer"
    Rectangle (0,330 640x30), "1st layer robot ID"
    Rectangle (0,360 640x30), "2nd layer robot ID"
    Rectangle (0,390 640x30), "3rd layer robot ID"
    Rectangle (0,420 640x30), "4th layer robot ID"
    Rectangle (0,450 640x30), "5th layer robot ID"
    Rectangle (0,480 640x30), "6th layer robot ID"
END_VISUALIZATION

// ---- Visualization/Shift register/Carton forming/CARTON_FORMING_SHIFT_ELEMENT.TcVIS
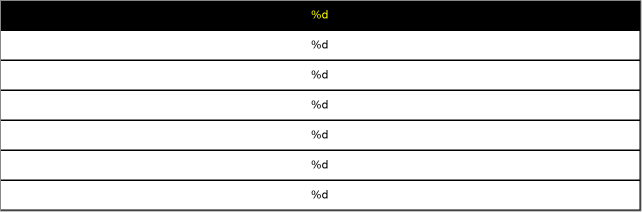
VISUALIZATION CARTON_FORMING_SHIFT_ELEMENT  // 642x212
VAR_INPUT
	index:		UDINT;
END_VAR
    Rectangle (0,0 640x30), "%d", text variable: wu_cartonForming_shiftRegister_debug.shift_debug[index].step_id
    Rectangle (0,30 640x30), "%d", text variable: wu_cartonForming_shiftRegister_debug.shift_debug[index].status.0, colour toggle: wu_cartonForming_shiftRegister_debug.shift_debug[index].status.0
    Rectangle (0,90 640x30), "%d", text variable: wu_cartonForming_shiftRegister_debug.shift_debug[index].reject_reason
    Rectangle (0,120 640x30), "%d", text variable: wu_cartonForming_shiftRegister_debug.shift_debug[index].status.4, colour toggle: wu_cartonForming_shiftRegister_debug.shift_debug[index].status.4
    Rectangle (0,180 640x30), "%d", text variable: wu_cartonForming_shiftRegister_debug.shift_debug[index].equipment_number
    Rectangle (0,150 640x30), "%d", text variable: wu_cartonForming_shiftRegister_debug.shift_debug[index].status.5, colour toggle: wu_cartonForming_shiftRegister_debug.shift_debug[index].status.5
    Rectangle (0,60 640x30), "%d", text variable: wu_cartonForming_shiftRegister_debug.shift_debug[index].status.1, colour toggle: wu_cartonForming_shiftRegister_debug.shift_debug[index].status.1
END_VISUALIZATION

// ---- Visualization/Shift register/Carton forming/CARTON_FORMING_SHIFT_ELEMENT_DESCRIPTION.TcVIS
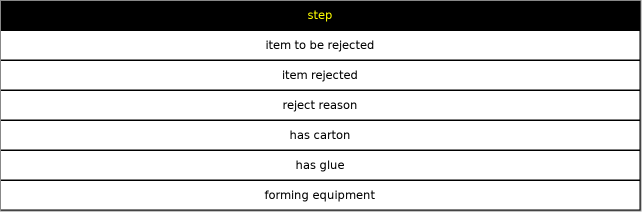
VISUALIZATION CARTON_FORMING_SHIFT_ELEMENT_DESCRIPTION  // 642x212
    Rectangle (0,0 640x30), "step"
    Rectangle (0,30 640x30), "item to be rejected"
    Rectangle (0,90 640x30), "reject reason"
    Rectangle (0,120 640x30), "has carton"
    Rectangle (0,180 640x30), "forming equipment"
    Rectangle (0,150 640x30), "has glue"
    Rectangle (0,60 640x30), "item rejected"
END_VISUALIZATION

// ---- Visualization/Shift register/Carton pickup/CARTON_PICKUP_SHIFT_ELEMENT_DESCRIPTION.TcVIS
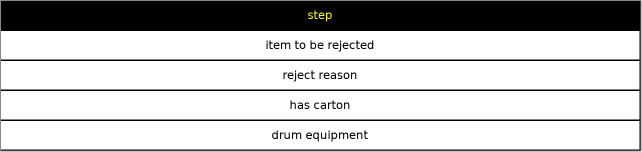
VISUALIZATION CARTON_PICKUP_SHIFT_ELEMENT_DESCRIPTION  // 642x152
    Rectangle (0,0 640x30), "step"
    Rectangle (0,30 640x30), "item to be rejected"
    Rectangle (0,60 640x30), "reject reason"
    Rectangle (0,90 640x30), "has carton"
    Rectangle (0,120 640x30), "drum equipment"
END_VISUALIZATION

// ---- Visualization/Shift register/Carton pickup/CARTON_PICKUP_SHIFT_ELEMENT.TcVIS
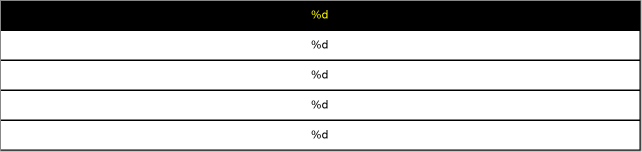
VISUALIZATION CARTON_PICKUP_SHIFT_ELEMENT  // 642x152
VAR_INPUT
	index:		UDINT;
END_VAR
    Rectangle (0,0 640x30), "%d", text variable: wu_cartonPickup_shiftRegister_debug.shift_debug[index].step_id
    Rectangle (0,30 640x30), "%d", text variable: wu_cartonPickup_shiftRegister_debug.shift_debug[index].status.0, colour toggle: wu_cartonPickup_shiftRegister_debug.shift_debug[index].status.0
    Rectangle (0,60 640x30), "%d", text variable: wu_cartonPickup_shiftRegister_debug.shift_debug[index].reject_reason
    Rectangle (0,90 640x30), "%d", text variable: wu_cartonPickup_shiftRegister_debug.shift_debug[index].status.4, colour toggle: wu_cartonPickup_shiftRegister_debug.shift_debug[index].status.4
    Rectangle (0,120 640x30), "%d", text variable: wu_cartonPickup_shiftRegister_debug.shift_debug[index].equipment_number
END_VISUALIZATION

// ---- Visualization/Shift register/CARTON_SHIFT.TcVIS
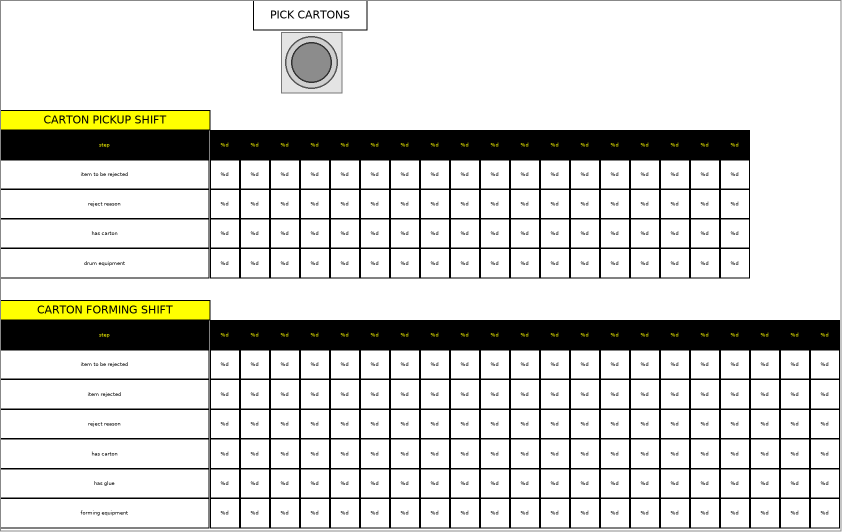
VISUALIZATION CARTON_SHIFT  // 842x532
    Frame (0,130 210x150)
        shows CARTON_PICKUP_SHIFT_ELEMENT_DESCRIPTION()
    Rectangle (0,110 210x20), "CARTON PICKUP SHIFT"
    Frame (210,130 30x150)
        shows CARTON_PICKUP_SHIFT_ELEMENT(index := 95)
    Frame (240,130 30x150)
        shows CARTON_PICKUP_SHIFT_ELEMENT(index := 96)
    Frame (270,130 30x150)
        shows CARTON_PICKUP_SHIFT_ELEMENT(index := 1)
    Frame (270,130 30x150)
        shows CARTON_PICKUP_SHIFT_ELEMENT(index := 97)
    Frame (300,130 30x150)
        shows CARTON_PICKUP_SHIFT_ELEMENT(index := 98)
    Frame (330,130 30x150)
        shows CARTON_PICKUP_SHIFT_ELEMENT(index := 1)
    Frame (330,130 30x150)
        shows CARTON_PICKUP_SHIFT_ELEMENT(index := 99)
    Frame (360,130 30x150)
        shows CARTON_PICKUP_SHIFT_ELEMENT(index := 100)
    Frame (390,130 30x150)
        shows CARTON_PICKUP_SHIFT_ELEMENT(index := 101)
    Frame (420,130 30x150)
        shows CARTON_PICKUP_SHIFT_ELEMENT(index := 102)
    Frame (450,130 30x150)
        shows CARTON_PICKUP_SHIFT_ELEMENT(index := 103)
    Frame (480,130 30x150)
        shows CARTON_PICKUP_SHIFT_ELEMENT(index := 104)
    Frame (510,130 30x150)
        shows CARTON_PICKUP_SHIFT_ELEMENT(index := 105)
    Frame (540,130 30x150)
        shows CARTON_PICKUP_SHIFT_ELEMENT(index := 106)
    Frame (570,130 30x150)
        shows CARTON_PICKUP_SHIFT_ELEMENT(index := 107)
    Frame (600,130 30x150)
        shows CARTON_PICKUP_SHIFT_ELEMENT(index := 108)
    Frame (630,130 30x150)
        shows CARTON_PICKUP_SHIFT_ELEMENT(index := 109)
    Frame (660,130 30x150)
        shows CARTON_PICKUP_SHIFT_ELEMENT(index := 110)
    Frame (690,130 30x150)
        shows CARTON_PICKUP_SHIFT_ELEMENT(index := 111)
    Frame (720,130 30x150)
        shows CARTON_PICKUP_SHIFT_ELEMENT(index := 112)
    Rectangle (0,300 210x20), "CARTON FORMING SHIFT"
    Frame (0,320 210x210)
        shows CARTON_FORMING_SHIFT_ELEMENT_DESCRIPTION()
    Frame (210,320 30x210)
        shows CARTON_FORMING_SHIFT_ELEMENT(index := 100)
    Frame (240,320 30x210)
        shows CARTON_FORMING_SHIFT_ELEMENT(index := 101)
    Frame (270,320 30x210)
        shows CARTON_FORMING_SHIFT_ELEMENT(index := 102)
    Frame (300,320 30x210)
        shows CARTON_FORMING_SHIFT_ELEMENT(index := 103)
    Frame (330,320 30x210)
        shows CARTON_FORMING_SHIFT_ELEMENT(index := 104)
    Frame (360,320 30x210)
        shows CARTON_FORMING_SHIFT_ELEMENT(index := 105)
    Frame (390,320 30x210)
        shows CARTON_FORMING_SHIFT_ELEMENT(index := 106)
    Frame (420,320 30x210)
        shows CARTON_FORMING_SHIFT_ELEMENT(index := 107)
    Frame (450,320 30x210)
        shows CARTON_FORMING_SHIFT_ELEMENT(index := 108)
    Frame (480,320 30x210)
        shows CARTON_FORMING_SHIFT_ELEMENT(index := 109)
    Frame (510,320 30x210)
        shows CARTON_FORMING_SHIFT_ELEMENT(index := 110)
    Frame (540,320 30x210)
        shows CARTON_FORMING_SHIFT_ELEMENT(index := 111)
    Frame (570,320 30x210)
        shows CARTON_FORMING_SHIFT_ELEMENT(index := 112)
    Frame (600,320 30x210)
        shows CARTON_FORMING_SHIFT_ELEMENT(index := 113)
    Frame (630,320 30x210)
        shows CARTON_FORMING_SHIFT_ELEMENT(index := 114)
    Frame (660,320 30x210)
        shows CARTON_FORMING_SHIFT_ELEMENT(index := 115)
    Frame (690,320 30x210)
        shows CARTON_FORMING_SHIFT_ELEMENT(index := 116)
    Frame (720,320 30x210)
        shows CARTON_FORMING_SHIFT_ELEMENT(index := 117)
    PushSwitch (279,32 65x61), variable: wu_cartonPickup_drums_suction.debug, behaviour: TOGGLE, style: Switch-PushSwitch-Gray
    Rectangle (253,0 114x30), "PICK CARTONS"
    Frame (750,320 30x210)
        shows CARTON_FORMING_SHIFT_ELEMENT(index := 118)
    Frame (780,320 30x210)
        shows CARTON_FORMING_SHIFT_ELEMENT(index := 119)
    Frame (810,320 30x210)
        shows CARTON_FORMING_SHIFT_ELEMENT(index := 120)
END_VISUALIZATION

// ---- Visualization/Shift register/Cups feeding/CUPS_FEEDING_SHIFT_ELEMENT.TcVIS
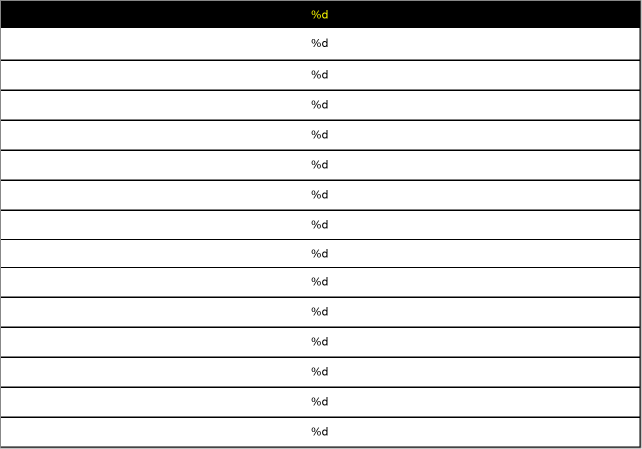
VISUALIZATION CUPS_FEEDING_SHIFT_ELEMENT  // 642x449
VAR_INPUT
	index:		UDINT;
END_VAR
    Rectangle (0,0 640x30), "%d", text variable: csp_case_main_statistics_debug.outer_shift_debug[index].step_id
    Rectangle (0,27 640x33), "%d", text variable: csp_case_main_statistics_debug.outer_shift_debug[index].status.1, colour toggle: csp_case_main_statistics_debug.outer_shift_debug[index].status.1
    Rectangle (0,150 640x30), "%d", text variable: csp_case_main_statistics_debug.outer_shift_debug[index].status.5, colour toggle: csp_case_main_statistics_debug.outer_shift_debug[index].status.5
    Rectangle (0,60 640x30), "%d", text variable: csp_case_main_statistics_debug.outer_shift_debug[index].reject_reason, colour toggle: csp_case_main_statistics_debug.outer_shift_debug[index].reject_reason
    Rectangle (0,180 640x30), "%d", text variable: csp_case_main_statistics_debug.outer_shift_debug[index].status.6, colour toggle: csp_case_main_statistics_debug.outer_shift_debug[index].status.6
    Rectangle (0,120 640x30), "%d", text variable: csp_case_main_statistics_debug.outer_shift_debug[index].status.4, colour toggle: csp_case_main_statistics_debug.outer_shift_debug[index].status.4
    Rectangle (0,210 640x30), "%d", text variable: csp_case_main_statistics_debug.outer_shift_debug[index].status.7, colour toggle: csp_case_main_statistics_debug.outer_shift_debug[index].status.7
    Rectangle (0,239 640x30), "%d", text variable: csp_case_main_statistics_debug.outer_shift_debug[index].status.8, colour toggle: csp_case_main_statistics_debug.outer_shift_debug[index].status.8
    Rectangle (0,267 640x30), "%d", text variable: csp_case_main_statistics_debug.outer_shift_debug[index].status.10, colour toggle: csp_case_main_statistics_debug.outer_shift_debug[index].status.10
    Rectangle (0,297 640x30), "%d", text variable: csp_case_main_statistics_debug.outer_shift_debug[index].status.11, colour toggle: csp_case_main_statistics_debug.outer_shift_debug[index].status.11
    Rectangle (0,327 640x30), "%d", text variable: csp_case_main_statistics_debug.outer_shift_debug[index].status.12, colour toggle: csp_case_main_statistics_debug.outer_shift_debug[index].status.12
    Rectangle (0,357 640x30), "%d", text variable: csp_case_main_statistics_debug.outer_shift_debug[index].status.13, colour toggle: csp_case_main_statistics_debug.outer_shift_debug[index].status.13
    Rectangle (0,387 640x30), "%d", text variable: csp_case_main_statistics_debug.outer_shift_debug[index].status.15, colour toggle: csp_case_main_statistics_debug.outer_shift_debug[index].status.15
    Rectangle (0,417 640x30), "%d", text variable: csp_transfer_main_statistics_debug.transfer_shift_debug[index].status.16, colour toggle: csp_transfer_main_statistics_debug.transfer_shift_debug[index].status.16
    Rectangle (0,90 640x30), "%d", text variable: csp_case_main_statistics_debug.outer_shift_debug[index].status.3, colour toggle: csp_case_main_statistics_debug.outer_shift_debug[index].status.3
END_VISUALIZATION

// ---- Visualization/Shift register/Cups feeding/CUPS_FEEDING_SHIFT_ELEMENT_DESCRIPTION.TcVIS
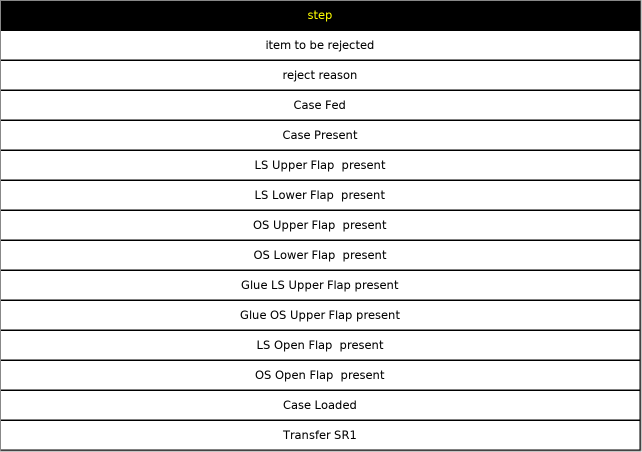
VISUALIZATION CUPS_FEEDING_SHIFT_ELEMENT_DESCRIPTION  // 642x452
    Rectangle (0,0 640x30), "step"
    Rectangle (0,30 640x30), "item to be rejected", tooltip "%d"
    Rectangle (0,60 640x30), "reject reason"
    Rectangle (0,90 640x30), "Case Fed"
    Rectangle (0,120 640x30), "Case Present"
    Rectangle (0,150 640x30), "LS Upper Flap present"
    Rectangle (0,180 640x30), "LS Lower Flap present"
    Rectangle (0,210 640x30), "OS Upper Flap present"
    Rectangle (0,240 640x30), "OS Lower Flap present"
    Rectangle (0,270 640x30), "Glue LS Upper Flap present"
    Rectangle (0,330 640x30), "LS Open Flap present"
    Rectangle (0,360 640x30), "OS Open Flap present"
    Rectangle (0,390 640x30), "Case Loaded"
    Rectangle (0,420 640x30), "Transfer SR1"
    Rectangle (0,300 640x30), "Glue OS Upper Flap present"
END_VISUALIZATION

// ---- Visualization/Shift register/CUPS_PICK_AND_PLACE.TcVIS
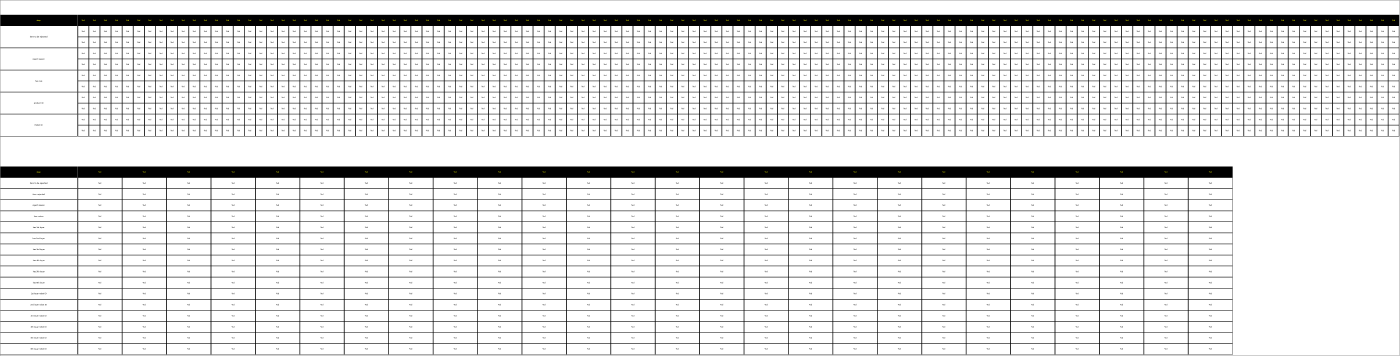
VISUALIZATION CUPS_PICK_AND_PLACE  // 3782x962
    Frame (210,40 30x330)
        shows TWISTED_CUPS_SHIFT_ELEMENT(index := 50)
    Frame (240,40 30x330)
        shows TWISTED_CUPS_SHIFT_ELEMENT(index := 51)
    Frame (270,40 30x330)
        shows TWISTED_CUPS_SHIFT_ELEMENT(index := 52)
    Frame (300,40 30x330)
        shows TWISTED_CUPS_SHIFT_ELEMENT(index := 53)
    Frame (330,40 30x330)
        shows TWISTED_CUPS_SHIFT_ELEMENT(index := 54)
    Frame (360,40 30x330)
        shows TWISTED_CUPS_SHIFT_ELEMENT(index := 55)
    Frame (390,40 30x330)
        shows TWISTED_CUPS_SHIFT_ELEMENT(index := 56)
    Frame (420,40 30x330)
        shows TWISTED_CUPS_SHIFT_ELEMENT(index := 57)
    Frame (450,40 30x330)
        shows TWISTED_CUPS_SHIFT_ELEMENT(index := 58)
    Frame (480,40 30x330)
        shows TWISTED_CUPS_SHIFT_ELEMENT(index := 59)
    Frame (510,40 30x330)
        shows TWISTED_CUPS_SHIFT_ELEMENT(index := 60)
    Frame (0,40 210x330)
        shows TWISTED_CUPS_SHIFT_ELEMENT_DESCRIPTION()
    Frame (540,40 30x330)
        shows TWISTED_CUPS_SHIFT_ELEMENT(index := 61)
    Frame (570,40 30x330)
        shows TWISTED_CUPS_SHIFT_ELEMENT(index := 62)
    Frame (600,40 30x330)
        shows TWISTED_CUPS_SHIFT_ELEMENT(index := 63)
    Frame (630,40 30x330)
        shows TWISTED_CUPS_SHIFT_ELEMENT(index := 64)
    Frame (660,40 30x330)
        shows TWISTED_CUPS_SHIFT_ELEMENT(index := 65)
    Frame (690,40 30x330)
        shows TWISTED_CUPS_SHIFT_ELEMENT(index := 66)
    Frame (720,40 30x330)
        shows TWISTED_CUPS_SHIFT_ELEMENT(index := 67)
    Frame (750,40 30x330)
        shows TWISTED_CUPS_SHIFT_ELEMENT(index := 68)
    Frame (780,40 30x330)
        shows TWISTED_CUPS_SHIFT_ELEMENT(index := 69)
    Frame (810,40 30x330)
        shows TWISTED_CUPS_SHIFT_ELEMENT(index := 70)
    Frame (840,40 30x330)
        shows TWISTED_CUPS_SHIFT_ELEMENT(index := 71)
    Frame (870,40 30x330)
        shows TWISTED_CUPS_SHIFT_ELEMENT(index := 72)
    Frame (900,40 30x330)
        shows TWISTED_CUPS_SHIFT_ELEMENT(index := 73)
    Frame (930,40 30x330)
        shows TWISTED_CUPS_SHIFT_ELEMENT(index := 74)
    Frame (960,40 30x330)
        shows TWISTED_CUPS_SHIFT_ELEMENT(index := 75)
    Frame (990,40 30x330)
        shows TWISTED_CUPS_SHIFT_ELEMENT(index := 76)
    Frame (1020,40 30x330)
        shows TWISTED_CUPS_SHIFT_ELEMENT(index := 77)
    Frame (1050,40 30x330)
        shows TWISTED_CUPS_SHIFT_ELEMENT(index := 78)
    Frame (1080,40 30x330)
        shows TWISTED_CUPS_SHIFT_ELEMENT(index := 79)
    Frame (1110,40 30x330)
        shows TWISTED_CUPS_SHIFT_ELEMENT(index := 80)
    Frame (1140,40 30x330)
        shows TWISTED_CUPS_SHIFT_ELEMENT(index := 81)
    Frame (1170,40 30x330)
        shows TWISTED_CUPS_SHIFT_ELEMENT(index := 82)
    Frame (1200,40 30x330)
        shows TWISTED_CUPS_SHIFT_ELEMENT(index := 83)
    Frame (1230,40 30x330)
        shows TWISTED_CUPS_SHIFT_ELEMENT(index := 84)
    Frame (1260,40 30x330)
        shows TWISTED_CUPS_SHIFT_ELEMENT(index := 85)
    Frame (1290,40 30x330)
        shows TWISTED_CUPS_SHIFT_ELEMENT(index := 86)
    Frame (1320,40 30x330)
        shows TWISTED_CUPS_SHIFT_ELEMENT(index := 87)
    Frame (1350,40 30x330)
        shows TWISTED_CUPS_SHIFT_ELEMENT(index := 88)
    Frame (1380,40 30x330)
        shows TWISTED_CUPS_SHIFT_ELEMENT(index := 89)
    Frame (1410,40 30x330)
        shows TWISTED_CUPS_SHIFT_ELEMENT(index := 90)
    Frame (1440,40 30x330)
        shows TWISTED_CUPS_SHIFT_ELEMENT(index := 91)
    Frame (1470,40 30x330)
        shows TWISTED_CUPS_SHIFT_ELEMENT(index := 92)
    Frame (1500,40 30x330)
        shows TWISTED_CUPS_SHIFT_ELEMENT(index := 93)
    Frame (1530,40 30x330)
        shows TWISTED_CUPS_SHIFT_ELEMENT(index := 94)
    Frame (1560,40 30x330)
        shows TWISTED_CUPS_SHIFT_ELEMENT(index := 95)
    Frame (1590,40 30x330)
        shows TWISTED_CUPS_SHIFT_ELEMENT(index := 96)
    Frame (1620,40 30x330)
        shows TWISTED_CUPS_SHIFT_ELEMENT(index := 97)
    Frame (1650,40 30x330)
        shows TWISTED_CUPS_SHIFT_ELEMENT(index := 98)
    Frame (1680,40 30x330)
        shows TWISTED_CUPS_SHIFT_ELEMENT(index := 99)
    Frame (1710,40 30x330)
        shows TWISTED_CUPS_SHIFT_ELEMENT(index := 100)
    Frame (1740,40 30x330)
        shows TWISTED_CUPS_SHIFT_ELEMENT(index := 101)
    Frame (1770,40 30x330)
        shows TWISTED_CUPS_SHIFT_ELEMENT(index := 102)
    Frame (1800,40 30x330)
        shows TWISTED_CUPS_SHIFT_ELEMENT(index := 103)
    Frame (1830,40 30x330)
        shows TWISTED_CUPS_SHIFT_ELEMENT(index := 104)
    Frame (1860,40 30x330)
        shows TWISTED_CUPS_SHIFT_ELEMENT(index := 105)
    Frame (1890,40 30x330)
        shows TWISTED_CUPS_SHIFT_ELEMENT(index := 106)
    Frame (1920,40 30x330)
        shows TWISTED_CUPS_SHIFT_ELEMENT(index := 107)
    Frame (1950,40 30x330)
        shows TWISTED_CUPS_SHIFT_ELEMENT(index := 108)
    Frame (1980,40 30x330)
        shows TWISTED_CUPS_SHIFT_ELEMENT(index := 109)
    Frame (2010,40 30x330)
        shows TWISTED_CUPS_SHIFT_ELEMENT(index := 110)
    Frame (2040,40 30x330)
        shows TWISTED_CUPS_SHIFT_ELEMENT(index := 111)
    Frame (2070,40 30x330)
        shows TWISTED_CUPS_SHIFT_ELEMENT(index := 112)
    Frame (2100,40 30x330)
        shows TWISTED_CUPS_SHIFT_ELEMENT(index := 113)
    Frame (2130,40 30x330)
        shows TWISTED_CUPS_SHIFT_ELEMENT(index := 114)
    Frame (2160,40 30x330)
        shows TWISTED_CUPS_SHIFT_ELEMENT(index := 115)
    Frame (2190,40 30x330)
        shows TWISTED_CUPS_SHIFT_ELEMENT(index := 116)
    Frame (2220,40 30x330)
        shows TWISTED_CUPS_SHIFT_ELEMENT(index := 117)
    Frame (2250,40 30x330)
        shows TWISTED_CUPS_SHIFT_ELEMENT(index := 118)
    Frame (2280,40 30x330)
        shows TWISTED_CUPS_SHIFT_ELEMENT(index := 119)
    Frame (2310,40 30x330)
        shows TWISTED_CUPS_SHIFT_ELEMENT(index := 120)
    Frame (0,450 210x510)
        shows CARTON_FILLING_SHIFT_ELEMENT_DESCRIPTION()
    Frame (2340,40 30x330)
        shows TWISTED_CUPS_SHIFT_ELEMENT(index := 121)
    Frame (2370,40 30x330)
        shows TWISTED_CUPS_SHIFT_ELEMENT(index := 122)
    Frame (2400,40 30x330)
        shows TWISTED_CUPS_SHIFT_ELEMENT(index := 123)
    Frame (2430,40 30x330)
        shows TWISTED_CUPS_SHIFT_ELEMENT(index := 124)
    Frame (2460,40 30x330)
        shows TWISTED_CUPS_SHIFT_ELEMENT(index := 125)
    Frame (2490,40 30x330)
        shows TWISTED_CUPS_SHIFT_ELEMENT(index := 126)
    Frame (2520,40 30x330)
        shows TWISTED_CUPS_SHIFT_ELEMENT(index := 127)
    Frame (2550,40 30x330)
        shows TWISTED_CUPS_SHIFT_ELEMENT(index := 128)
    Frame (2580,40 30x330)
        shows TWISTED_CUPS_SHIFT_ELEMENT(index := 129)
    Frame (2610,40 30x330)
        shows TWISTED_CUPS_SHIFT_ELEMENT(index := 130)
    Frame (2640,40 30x330)
        shows TWISTED_CUPS_SHIFT_ELEMENT(index := 131)
    Frame (2670,40 30x330)
        shows TWISTED_CUPS_SHIFT_ELEMENT(index := 132)
    Frame (2700,40 30x330)
        shows TWISTED_CUPS_SHIFT_ELEMENT(index := 133)
    Frame (2730,40 30x330)
        shows TWISTED_CUPS_SHIFT_ELEMENT(index := 134)
    Frame (2760,40 30x330)
        shows TWISTED_CUPS_SHIFT_ELEMENT(index := 135)
    Frame (2790,40 30x330)
        shows TWISTED_CUPS_SHIFT_ELEMENT(index := 136)
    Frame (2820,40 30x330)
        shows TWISTED_CUPS_SHIFT_ELEMENT(index := 137)
    Frame (2850,40 30x330)
        shows TWISTED_CUPS_SHIFT_ELEMENT(index := 138)
    Frame (2880,40 30x330)
        shows TWISTED_CUPS_SHIFT_ELEMENT(index := 139)
    Frame (2910,40 30x330)
        shows TWISTED_CUPS_SHIFT_ELEMENT(index := 140)
    Frame (2940,40 30x330)
        shows TWISTED_CUPS_SHIFT_ELEMENT(index := 141)
    Frame (2970,40 30x330)
        shows TWISTED_CUPS_SHIFT_ELEMENT(index := 142)
    Frame (3000,40 30x330)
        shows TWISTED_CUPS_SHIFT_ELEMENT(index := 143)
    Frame (3030,40 30x330)
        shows TWISTED_CUPS_SHIFT_ELEMENT(index := 144)
    Frame (3060,40 30x330)
        shows TWISTED_CUPS_SHIFT_ELEMENT(index := 145)
    Frame (3090,40 30x330)
        shows TWISTED_CUPS_SHIFT_ELEMENT(index := 146)
    Frame (3120,40 30x330)
        shows TWISTED_CUPS_SHIFT_ELEMENT(index := 147)
    Frame (3150,40 30x330)
        shows TWISTED_CUPS_SHIFT_ELEMENT(index := 148)
    Frame (3180,40 30x330)
        shows TWISTED_CUPS_SHIFT_ELEMENT(index := 149)
    Frame (3210,40 30x330)
        shows TWISTED_CUPS_SHIFT_ELEMENT(index := 150)
    Frame (3240,40 30x330)
        shows TWISTED_CUPS_SHIFT_ELEMENT(index := 151)
    Frame (3270,40 30x330)
        shows TWISTED_CUPS_SHIFT_ELEMENT(index := 152)
    Frame (3300,40 30x330)
        shows TWISTED_CUPS_SHIFT_ELEMENT(index := 153)
    Frame (3330,40 30x330)
        shows TWISTED_CUPS_SHIFT_ELEMENT(index := 154)
    Frame (3360,40 30x330)
        shows TWISTED_CUPS_SHIFT_ELEMENT(index := 155)
    Frame (3390,40 30x330)
        shows TWISTED_CUPS_SHIFT_ELEMENT(index := 156)
    Frame (3420,40 30x330)
        shows TWISTED_CUPS_SHIFT_ELEMENT(index := 157)
    Frame (3450,40 30x330)
        shows TWISTED_CUPS_SHIFT_ELEMENT(index := 158)
    Frame (3480,40 30x330)
        shows TWISTED_CUPS_SHIFT_ELEMENT(index := 159)
    Frame (3510,40 30x330)
        shows TWISTED_CUPS_SHIFT_ELEMENT(index := 160)
    Frame (3540,40 30x330)
        shows TWISTED_CUPS_SHIFT_ELEMENT(index := 161)
    Frame (3570,40 30x330)
        shows TWISTED_CUPS_SHIFT_ELEMENT(index := 162)
    Frame (3600,40 30x330)
        shows TWISTED_CUPS_SHIFT_ELEMENT(index := 163)
    Frame (3630,40 30x330)
        shows TWISTED_CUPS_SHIFT_ELEMENT(index := 164)
    Frame (3660,40 30x330)
        shows TWISTED_CUPS_SHIFT_ELEMENT(index := 165)
    Frame (3690,40 30x330)
        shows TWISTED_CUPS_SHIFT_ELEMENT(index := 166)
    Frame (3720,40 30x330)
        shows TWISTED_CUPS_SHIFT_ELEMENT(index := 167)
    Frame (3750,40 30x330)
        shows TWISTED_CUPS_SHIFT_ELEMENT(index := 168)
    Frame (210,450 120x510)
        shows CARTON_FILLING_SHIFT_ELEMENT(index := 135)
    Frame (330,450 120x510)
        shows CARTON_FILLING_SHIFT_ELEMENT(index := 134)
    Frame (450,450 120x510)
        shows CARTON_FILLING_SHIFT_ELEMENT(index := 133)
    Frame (570,450 120x510)
        shows CARTON_FILLING_SHIFT_ELEMENT(index := 132)
    Frame (690,450 120x510)
        shows CARTON_FILLING_SHIFT_ELEMENT(index := 131)
    Frame (810,450 120x510)
        shows CARTON_FILLING_SHIFT_ELEMENT(index := 130)
    Frame (930,450 120x510)
        shows CARTON_FILLING_SHIFT_ELEMENT(index := 129)
    Frame (1050,450 120x510)
        shows CARTON_FILLING_SHIFT_ELEMENT(index := 128)
    Frame (1170,450 120x510)
        shows CARTON_FILLING_SHIFT_ELEMENT(index := 127)
    Frame (1290,450 120x510)
        shows CARTON_FILLING_SHIFT_ELEMENT(index := 126)
    Frame (1410,450 120x510)
        shows CARTON_FILLING_SHIFT_ELEMENT(index := 125)
    Frame (1530,450 120x510)
        shows CARTON_FILLING_SHIFT_ELEMENT(index := 124)
    Frame (1650,450 120x510)
        shows CARTON_FILLING_SHIFT_ELEMENT(index := 123)
    Frame (1770,450 120x510)
        shows CARTON_FILLING_SHIFT_ELEMENT(index := 122)
    Frame (1890,450 120x510)
        shows CARTON_FILLING_SHIFT_ELEMENT(index := 121)
    Frame (2010,450 120x510)
        shows CARTON_FILLING_SHIFT_ELEMENT(index := 120)
    Frame (2130,450 120x510)
        shows CARTON_FILLING_SHIFT_ELEMENT(index := 119)
    Frame (2250,450 120x510)
        shows CARTON_FILLING_SHIFT_ELEMENT(index := 118)
    Frame (2370,450 120x510)
        shows CARTON_FILLING_SHIFT_ELEMENT(index := 117)
    Frame (2490,450 120x510)
        shows CARTON_FILLING_SHIFT_ELEMENT(index := 116)
    Frame (2610,450 120x510)
        shows CARTON_FILLING_SHIFT_ELEMENT(index := 115)
    Frame (2730,450 120x510)
        shows CARTON_FILLING_SHIFT_ELEMENT(index := 114)
    Frame (2850,450 120x510)
        shows CARTON_FILLING_SHIFT_ELEMENT(index := 113)
    Frame (2970,450 120x510)
        shows CARTON_FILLING_SHIFT_ELEMENT(index := 112)
    Frame (3090,450 120x510)
        shows CARTON_FILLING_SHIFT_ELEMENT(index := 111)
    Frame (3210,450 120x510)
        shows CARTON_FILLING_SHIFT_ELEMENT(index := 110)
END_VISUALIZATION

// ---- Visualization/Shift register/CUPS_SHIFT.TcVIS
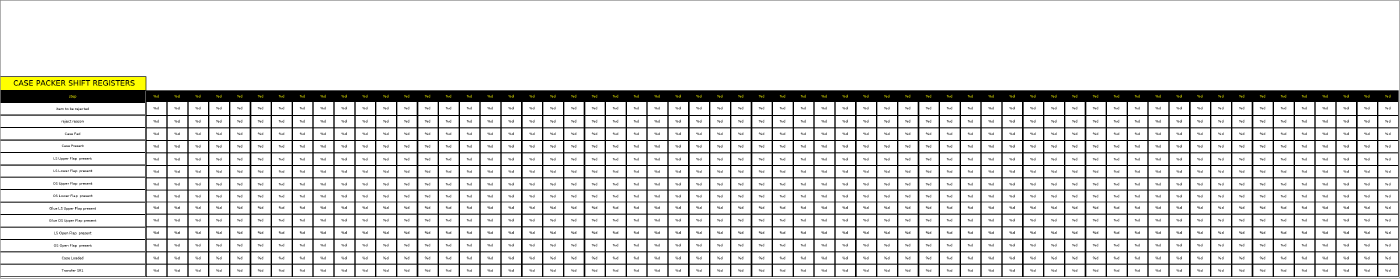
VISUALIZATION CUPS_SHIFT  // 2012x402
    Frame (0,130 210x270)
        shows CUPS_FEEDING_SHIFT_ELEMENT_DESCRIPTION()
    Rectangle (0,110 210x20), "CASE PACKER SHIFT REGISTERS"
    Frame (390,130 30x270)
        shows CUPS_FEEDING_SHIFT_ELEMENT(index := 7)
        shows CUPS_FEEDING_SHIFT_ELEMENT()
    Frame (420,130 30x270)
        shows CUPS_FEEDING_SHIFT_ELEMENT(index := 8)
    Frame (450,130 30x270)
        shows CUPS_FEEDING_SHIFT_ELEMENT(index := 9)
    Frame (480,130 30x270)
        shows CUPS_FEEDING_SHIFT_ELEMENT(index := 10)
    Frame (510,130 30x270)
        shows CUPS_FEEDING_SHIFT_ELEMENT(index := 11)
    Frame (540,130 30x270)
        shows CUPS_FEEDING_SHIFT_ELEMENT(index := 12)
    Frame (570,130 30x270)
        shows CUPS_FEEDING_SHIFT_ELEMENT(index := 13)
    Frame (600,130 30x270)
        shows CUPS_FEEDING_SHIFT_ELEMENT(index := 14)
    Frame (630,130 30x270)
        shows CUPS_FEEDING_SHIFT_ELEMENT(index := 15)
    Frame (660,130 30x270)
        shows CUPS_FEEDING_SHIFT_ELEMENT(index := 16)
    Frame (690,130 30x270)
        shows CUPS_FEEDING_SHIFT_ELEMENT(index := 17)
    Frame (720,130 30x270)
        shows CUPS_FEEDING_SHIFT_ELEMENT(index := 18)
    Frame (750,130 30x270)
        shows CUPS_FEEDING_SHIFT_ELEMENT(index := 19)
    Frame (780,130 30x270)
        shows CUPS_FEEDING_SHIFT_ELEMENT(index := 20)
    Frame (810,130 30x270)
        shows CUPS_FEEDING_SHIFT_ELEMENT(index := 21)
    Frame (840,130 30x270)
        shows CUPS_FEEDING_SHIFT_ELEMENT(index := 22)
    Frame (870,130 30x270)
        shows CUPS_FEEDING_SHIFT_ELEMENT(index := 23)
    Frame (900,130 30x270)
        shows CUPS_FEEDING_SHIFT_ELEMENT(index := 24)
    Frame (930,130 30x270)
        shows CUPS_FEEDING_SHIFT_ELEMENT(index := 25)
    Frame (960,130 30x270)
        shows CUPS_FEEDING_SHIFT_ELEMENT(index := 26)
    Frame (990,130 30x270)
        shows CUPS_FEEDING_SHIFT_ELEMENT(index := 27)
    Frame (1020,130 30x270)
        shows CUPS_FEEDING_SHIFT_ELEMENT(index := 28)
    Frame (1050,130 30x270)
        shows CUPS_FEEDING_SHIFT_ELEMENT(index := 29)
    Frame (1080,130 30x270)
        shows CUPS_FEEDING_SHIFT_ELEMENT(index := 30)
    Frame (1110,130 30x270)
        shows CUPS_FEEDING_SHIFT_ELEMENT(index := 31)
    Frame (1140,130 30x270)
        shows CUPS_FEEDING_SHIFT_ELEMENT(index := 32)
    Frame (1170,130 30x270)
        shows CUPS_FEEDING_SHIFT_ELEMENT(index := 33)
    Frame (1200,130 30x270)
        shows CUPS_FEEDING_SHIFT_ELEMENT(index := 34)
    Frame (1230,130 30x270)
        shows CUPS_FEEDING_SHIFT_ELEMENT(index := 35)
    Frame (1260,130 30x270)
        shows CUPS_FEEDING_SHIFT_ELEMENT(index := 36)
    Frame (1290,130 30x270)
        shows CUPS_FEEDING_SHIFT_ELEMENT(index := 37)
    Frame (1320,130 30x270)
        shows CUPS_FEEDING_SHIFT_ELEMENT(index := 38)
    Frame (1350,130 30x270)
        shows CUPS_FEEDING_SHIFT_ELEMENT(index := 39)
    Frame (1380,130 30x270)
        shows CUPS_FEEDING_SHIFT_ELEMENT(index := 40)
    Frame (1410,130 30x270)
        shows CUPS_FEEDING_SHIFT_ELEMENT(index := 41)
    Frame (1440,130 30x270)
        shows CUPS_FEEDING_SHIFT_ELEMENT(index := 42)
    Frame (1470,130 30x270)
        shows CUPS_FEEDING_SHIFT_ELEMENT(index := 43)
    Frame (1500,130 30x270)
        shows CUPS_FEEDING_SHIFT_ELEMENT(index := 44)
    Frame (1530,130 30x270)
        shows CUPS_FEEDING_SHIFT_ELEMENT(index := 45)
    Frame (1560,130 30x270)
        shows CUPS_FEEDING_SHIFT_ELEMENT(index := 46)
    Frame (1590,130 30x270)
        shows CUPS_FEEDING_SHIFT_ELEMENT(index := 47)
    Frame (1620,130 30x270)
        shows CUPS_FEEDING_SHIFT_ELEMENT(index := 48)
    Frame (1650,130 30x270)
        shows CUPS_FEEDING_SHIFT_ELEMENT(index := 49)
    Frame (1680,130 30x270)
        shows CUPS_FEEDING_SHIFT_ELEMENT(index := 50)
    Frame (1710,130 30x270)
        shows CUPS_FEEDING_SHIFT_ELEMENT(index := 51)
    Frame (1740,130 30x270)
        shows CUPS_FEEDING_SHIFT_ELEMENT(index := 52)
    Frame (1770,130 30x270)
        shows CUPS_FEEDING_SHIFT_ELEMENT(index := 53)
    Frame (1800,130 30x270)
        shows CUPS_FEEDING_SHIFT_ELEMENT(index := 54)
    Frame (1830,130 30x270)
        shows CUPS_FEEDING_SHIFT_ELEMENT(index := 55)
    Frame (1860,130 30x270)
        shows CUPS_FEEDING_SHIFT_ELEMENT(index := 56)
    Frame (1890,130 30x270)
        shows CUPS_FEEDING_SHIFT_ELEMENT(index := 57)
    Frame (1920,130 30x270)
        shows CUPS_FEEDING_SHIFT_ELEMENT(index := 58)
    Frame (1950,130 30x270)
        shows CUPS_FEEDING_SHIFT_ELEMENT(index := 59)
    Frame (1980,130 30x270)
        shows CUPS_FEEDING_SHIFT_ELEMENT(index := 60)
    Frame (210,130 30x270)
        shows CUPS_FEEDING_SHIFT_ELEMENT(index := 1)
        shows CUPS_FEEDING_SHIFT_ELEMENT()
    Frame (240,130 30x270)
        shows CUPS_FEEDING_SHIFT_ELEMENT(index := 2)
        shows CUPS_FEEDING_SHIFT_ELEMENT()
    Frame (270,130 30x270)
        shows CUPS_FEEDING_SHIFT_ELEMENT(index := 3)
        shows CUPS_FEEDING_SHIFT_ELEMENT()
    Frame (300,130 30x270)
        shows CUPS_FEEDING_SHIFT_ELEMENT(index := 4)
        shows CUPS_FEEDING_SHIFT_ELEMENT()
    Frame (330,130 30x270)
        shows CUPS_FEEDING_SHIFT_ELEMENT(index := 5)
        shows CUPS_FEEDING_SHIFT_ELEMENT()
    Frame (360,130 30x270)
        shows CUPS_FEEDING_SHIFT_ELEMENT(index := 6)
        shows CUPS_FEEDING_SHIFT_ELEMENT()
END_VISUALIZATION

// ---- Visualization/Shift register/Twisted cups/TWISTED_CUPS_SHIFT_ELEMENT.TcVIS
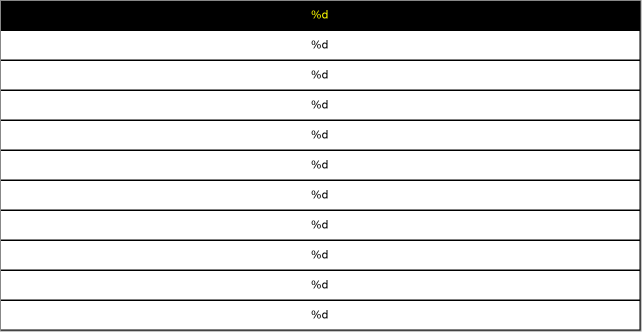
VISUALIZATION TWISTED_CUPS_SHIFT_ELEMENT  // 642x332
VAR_INPUT
	index:		UDINT;
END_VAR
    Rectangle (0,0 640x30), "%d", text variable: wu_twistedCups_shiftRegister_debug.outer_shift_debug[90+index].step_id
    Rectangle (0,30 640x30), "%d", text variable: wu_twistedCups_shiftRegister_debug.outer_shift_debug[90+index].status.0, colour toggle: wu_twistedCups_shiftRegister_debug.outer_shift_debug[90+index].status.0
    Rectangle (0,90 640x30), "%d", text variable: wu_twistedCups_shiftRegister_debug.outer_shift_debug[90+index].reject_reason
    Rectangle (0,150 640x30), "%d", text variable: wu_twistedCups_shiftRegister_debug.outer_shift_debug[90+index].status.3, colour toggle: wu_twistedCups_shiftRegister_debug.outer_shift_debug[90+index].status.3
    Rectangle (0,210 640x30), "%d", text variable: wu_twistedCups_shiftRegister_debug.outer_shift_debug[90+index].product_id
    Rectangle (0,60 640x30), "%d", text variable: wu_twistedCups_shiftRegister_debug.inner_shift_debug[90+index].status.0, colour toggle: wu_twistedCups_shiftRegister_debug.inner_shift_debug[90+index].status.0
    Rectangle (0,120 640x30), "%d", text variable: wu_twistedCups_shiftRegister_debug.inner_shift_debug[90+index].reject_reason
    Rectangle (0,180 640x30), "%d", text variable: wu_twistedCups_shiftRegister_debug.inner_shift_debug[90+index].status.3, colour toggle: wu_twistedCups_shiftRegister_debug.inner_shift_debug[90+index].status.3
    Rectangle (0,240 640x30), "%d", text variable: wu_twistedCups_shiftRegister_debug.inner_shift_debug[90+index].product_id
    Rectangle (0,270 640x30), "%d", text variable: wu_twistedCups_shiftRegister_debug.outer_shift_debug[90+index].robot_id
    Rectangle (0,300 640x30), "%d", text variable: wu_twistedCups_shiftRegister_debug.inner_shift_debug[90+index].robot_id
END_VISUALIZATION

// ---- Visualization/Shift register/Twisted cups/TWISTED_CUPS_SHIFT_ELEMENT_DESCRIPTION.TcVIS
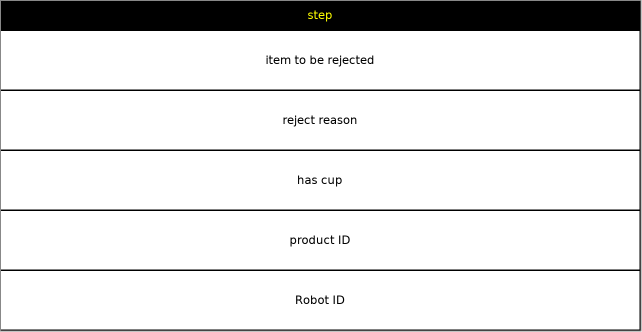
VISUALIZATION TWISTED_CUPS_SHIFT_ELEMENT_DESCRIPTION  // 642x332
    Rectangle (0,0 640x30), "step"
    Rectangle (0,30 640x60), "item to be rejected"
    Rectangle (0,90 640x60), "reject reason"
    Rectangle (0,150 640x60), "has cup"
    Rectangle (0,210 640x60), "product ID"
    Rectangle (0,270 640x60), "Robot ID"
END_VISUALIZATION
